PROGRAM PRG_TEST
VAR
	fbCheckPartTest		: FB_CellCheckPart_Test;
END_VAR

TcUnit.RUN();

END_PROGRAM

(* stored: Version 1.1.0.1, ProductVersion 3.1.4024.12
   POU PRG_TEST: Id {6c3deb47-32e2-470c-b370-1746d2072dba}, SpecialFunc None *)
